FUNCTION_BLOCK FB_RecipeBase IMPLEMENTS I_RecipeBuilder 

VAR
    _Config                 : ST_RecipeBuilder_Config;
	_ConfigProvider 		: I_GantryConfigProvider;

	
	
	_Limits : ST_Recipe_Limits;

    // --- NOWE ZMIENNE DO PRZECHOWYWANIA SEGMENTÓW ---
    _SegmentsCutX           : ARRAY [1..100] OF ST_CutSegment;
    _SegmentsCutY           : ARRAY [1..100] OF ST_CutSegment;
    _SegmentsGroove         : ARRAY [1..100] OF ST_CutSegment;
	_HolesDrill 			: ARRAY [1..100] OF ST_PointXY;
	_ShapeStart         	: ARRAY [1..100] OF ST_PointXY;
	_ShapesCount        	: INT := 1;
    _CurrentShapeIndex  	: INT := 1;
	_HolesToDrill   		: INT;
    _SegmentsToCutX         : INT;
    _SegmentsToCutY         : INT;
    _SegmentsToGroove       : INT;
	_FootprintX 			: REAL;
	_FootprintY 			: REAL;
	_MaxCopiesX				: DINT;
	_MaxCopiesY				: DINT;
	_ActualCopiesX			: DINT;
	_ActualCopiesY			: DINT;
	_NominalX 				: REAL;
    _NominalY 				: REAL;
	_Busy					: BOOL;
	_Done					: BOOL;
	_Error					: BOOL;
	
	// --- GENERYCZNY GENERATOR G-CODE (NCI) ---
    fbCreateFile    : ItpPpgCreateMain;
    fbAppendLine    : ItpPpgAppendGenericBlock;
    fbCloseFile     : ItpPpgCloseMain;
    
    _aGCodeBuffer   : ARRAY[1..600] OF STRING(255); 
    _nLinesToWrite  : INT;                          // Ile linii z bufora zapisać
    _nFileWriteStep : INT := 0;                     // Krok maszyny stanów zapisu
    _sGCodeFilePath : STRING(255);                  // Ścieżka pliku
	
	_GeometryWriter : I_GeometryWriter;
	
END_VAR

PROPERTY ActualCopiesX : DINT
GET
ActualCopiesX := _Config.RequestedCopiesX;
END_GET
END_PROPERTY

PROPERTY ActualCopiesY : DINT
GET
ActualCopiesY := _Config.RequestedCopiesY;
END_GET
END_PROPERTY

METHOD Build : BOOL
Build := FALSE;
END_METHOD

PROPERTY Busy : BOOL
GET
Busy := _Busy;
END_GET
SET
_Busy := Busy;
END_SET
END_PROPERTY

METHOD PROTECTED CalculateFootprint
VAR_INPUT
END_VAR
// Domyślny wymiar detalu (bez dodatków)
_NominalX := _Config.PanelFrontWidth;
_NominalY := _Config.PanelFrontLength;
END_METHOD

PROPERTY Config : ST_RecipeBuilder_Config
GET
Config := _Config;
END_GET
SET
VAR
    sTempGCodePath : STRING(255);
END_VAR
// 1. NAJPIERW robimy kopię tego co mamy w pamięci sterownika
sTempGCodePath := THIS^._Config.GCodePath; 

// 2. TERAZ przyjmujemy nową strukturę z HMI
_Config := Config;

// 3. PRZYWRACAMY ścieżkę do pliku
_Config.GCodePath := sTempGCodePath;

_Config.PanelFrontLength     := LIMIT(_Limits.PanelFrontLength.MinVal, Config.PanelFrontLength, _Limits.PanelFrontLength.MaxVal);
_Config.PanelFrontWidth      := LIMIT(_Limits.PanelFrontWidth.MinVal,  Config.PanelFrontWidth,  _Limits.PanelFrontWidth.MaxVal);
_Config.PanelHeight          := LIMIT(_Limits.PanelHeight.MinVal,      Config.PanelHeight,      _Limits.PanelHeight.MaxVal);
_Config.RailHeightCorrection := LIMIT(_Limits.RailHeightCorrection.MinVal, Config.RailHeightCorrection, _Limits.RailHeightCorrection.MaxVal);
_Config.GrooveDepthZ		 :=	LIMIT(_Limits.GrooveDepthZ.MinVal,	Config.GrooveDepthZ, _Limits.GrooveDepthZ.MaxVal);
_Config.Diameter 			 := LIMIT(_Limits.Diameter.MinVal, Config.Diameter, _Limits.Diameter.MaxVal);

_Config.CuttingOverpass      := LIMIT(_Limits.CuttingOverpass.MinVal, Config.CuttingOverpass, _Limits.CuttingOverpass.MaxVal);
_Config.GroovingOverpass     := LIMIT(_Limits.GroovingOverpass.MinVal, Config.GroovingOverpass, _Limits.GroovingOverpass.MaxVal);
_Config.Radius               := LIMIT(_Limits.Radius.MinVal, Config.Radius, _Limits.Radius.MaxVal);

THIS^.UpdateNestingLimits();


IF _Config.FillAll THEN
    _Config.RequestedCopiesX := _MaxCopiesX;
    _Config.RequestedCopiesY := _MaxCopiesY;
ELSE
    _Config.RequestedCopiesX := LIMIT(1, _Config.RequestedCopiesX, _MaxCopiesX);
    _Config.RequestedCopiesY := LIMIT(1, _Config.RequestedCopiesY, _MaxCopiesY);
END_IF
END_SET
END_PROPERTY

PROPERTY ConfigProvider : I_GantryConfigProvider
GET
ConfigProvider := _ConfigProvider;
END_GET
SET
_ConfigProvider := ConfigProvider;
END_SET
END_PROPERTY

PROPERTY CurrentShapeIndex : INT
GET
CurrentShapeIndex := _CurrentShapeIndex;
END_GET
SET
_CurrentShapeIndex := CurrentShapeIndex;
END_SET
END_PROPERTY

PROPERTY Done : BOOL
GET
Done := _Done;
END_GET
SET
_Done := Done;
END_SET
END_PROPERTY

PROPERTY Error : BOOL
GET
Error := _Error;
END_GET
SET
_Error := Error;
END_SET
END_PROPERTY

PROPERTY ExecutionRoute : E_ExecutionRoute
GET
END_GET
END_PROPERTY

PROPERTY FootprintX : REAL
GET
FootprintX := _FootprintX;
END_GET
SET
_FootprintX := FootprintX;
END_SET
END_PROPERTY

PROPERTY FootprintY : REAL
GET
FootprintY := _FootprintY;
END_GET
SET
_FootprintY := FootprintY;
END_SET
END_PROPERTY

PROPERTY GeometryWriter : I_GeometryWriter
GET
GeometryWriter := _GeometryWriter;
END_GET
SET
_GeometryWriter := GeometryWriter;
END_SET
END_PROPERTY

PROPERTY HolesDrill : REFERENCE TO ARRAY [1..100] OF ST_PointXY
GET
HolesDrill REF= _HolesDrill;
END_GET
END_PROPERTY

PROPERTY HolesToDrill : INT
GET
HolesToDrill := _HolesToDrill;
END_GET
END_PROPERTY

PROPERTY Limits : ST_Recipe_Limits
GET
Limits := _Limits;
END_GET
END_PROPERTY

PROPERTY MaxCopiesX : DINT
GET
MaxCopiesX := _MaxCopiesX;
END_GET
END_PROPERTY

PROPERTY MaxCopiesY : DINT
GET
MaxCopiesY := _MaxCopiesY ;
END_GET
END_PROPERTY

PROPERTY SegmentsCutX : REFERENCE TO ARRAY [1..100] OF ST_CutSegment
GET
SegmentsCutX REF= _SegmentsCutX;
END_GET
END_PROPERTY

PROPERTY SegmentsCutY : REFERENCE TO ARRAY [1..100] OF ST_CutSegment
GET
SegmentsCutY REF= _SegmentsCutY;
END_GET
END_PROPERTY

PROPERTY SegmentsGroove : REFERENCE TO ARRAY [1..100] OF ST_CutSegment
GET
SegmentsGroove REF= _SegmentsGroove;
END_GET
END_PROPERTY


PROPERTY SegmentsToCutX : INT
GET
SegmentsToCutX := _SegmentsToCutX;
END_GET
END_PROPERTY


PROPERTY SegmentsToCutY : INT
GET
SegmentsToCutY := _SegmentsToCutY;
END_GET
END_PROPERTY


PROPERTY SegmentsToGroove : INT
GET
SegmentsToGroove := _SegmentsToGroove;
END_GET
END_PROPERTY

PROPERTY ShapesCount : INT
GET
ShapesCount := _ShapesCount;
END_GET
END_PROPERTY

PROPERTY ShapeStart : REFERENCE TO ARRAY [1..100] OF ST_PointXY
GET
ShapeStart REF= _ShapeStart;
END_GET
END_PROPERTY

METHOD PUBLIC UpdateNestingLimits
VAR
    MaxOverpass     : REAL;
    MachineConfig   : ST_GantryXYZ_Config; // Zmienna do odczytu offsetu
    EffectiveBoardX : REAL;
    EffectiveBoardY : REAL;
END_VAR
VAR_INST
    bLogFired       : BOOL; // <-- Zapamięta, czy log już poszedł
END_VAR
// 1. Czysty gabaryt z logiki receptury
THIS^.CalculateFootprint();
MaxOverpass := MAX(_Config.CuttingOverpass, _Config.GroovingOverpass);
_FootprintX := _NominalX + (2.0 * MaxOverpass);
_FootprintY := _NominalY + (2.0 * MaxOverpass);

// 2. Pobranie Global Offsetu ORAZ wymiarów płyty z maszyny
IF _ConfigProvider <> 0 THEN
    MachineConfig := _ConfigProvider.Config;
ELSE
    // Awaryjny "fallback" jeśli Provider nie jest wstrzyknięty (np. w starych testach)
    MachineConfig.GlobalOffsetX := 0.0;
    MachineConfig.GlobalOffsetY := 0.0;
    MachineConfig.RawBoardX := 1220.0; // Domyślna płyta 
    MachineConfig.RawBoardY := 2440.0; // Domyślna płyta
	MachineConfig.RawBoardZ := 9.0;
END_IF

// 3. Efektywna wielkość płyty = Fizyczna płyta (z maszyny) minus offset początkowy
EffectiveBoardX := MachineConfig.RawBoardX - MachineConfig.GlobalOffsetX;
EffectiveBoardY := MachineConfig.RawBoardY - MachineConfig.GlobalOffsetY;

// 4. Przeliczanie kopii nestingu (zabezpieczenie na ujemne wymiary)
IF _FootprintX > 0.0 AND EffectiveBoardX > 0.0 THEN
    _MaxCopiesX := REAL_TO_DINT(TRUNC(EffectiveBoardX / _FootprintX));
ELSE
    _MaxCopiesX := 0;
END_IF

IF _FootprintY > 0.0 AND EffectiveBoardY > 0.0 THEN
    _MaxCopiesY := REAL_TO_DINT(TRUNC(EffectiveBoardY / _FootprintY));
ELSE
    _MaxCopiesY := 0;
END_IF

// =========================================================
// 5. WERYFIKACJA GABARYTÓW (Zabezpieczenie przed za dużym detalem)
// =========================================================
_Config.IsValid := (_MaxCopiesX > 0) AND (_MaxCopiesY > 0) AND (_NominalX > 0) AND (_NominalY > 0);

IF NOT _Config.IsValid THEN
    IF NOT bLogFired THEN
        ADSLOGSTR(ADSLOG_MSGTYPE_ERROR, 'UpdateNestingLimits: Konfiguracja odrzucona (IsValid = FALSE)! Sprawdzam dlaczego...', '');
        
        IF _MaxCopiesX <= 0 THEN 
            ADSLOGSTR(ADSLOG_MSGTYPE_ERROR, 'Powod: _MaxCopiesX <= 0 (Detal wychodzi poza szerokosc stolu)', ''); 
        END_IF
        IF _MaxCopiesY <= 0 THEN 
            ADSLOGSTR(ADSLOG_MSGTYPE_ERROR, 'Powod: _MaxCopiesY <= 0 (Detal wychodzi poza dlugosc stolu)', ''); 
        END_IF
        IF _NominalX <= 0 THEN 
            ADSLOGSTR(ADSLOG_MSGTYPE_ERROR, 'Powod: _NominalX <= 0 (Szerokosc Nominalna to zero!)', ''); 
        END_IF
        IF _NominalY <= 0 THEN 
            ADSLOGSTR(ADSLOG_MSGTYPE_ERROR, 'Powod: _NominalY <= 0 (Dlugosc Nominalna to zero!)', ''); 
        END_IF
        
        bLogFired := TRUE; // Zablokuj kolejne wysyłanie
    END_IF
ELSE
    // Jeśli znowu jest poprawnie (np. poprawiono na HMI), odblokuj logi na przyszłość
    bLogFired := FALSE;
END_IF

// =========================================================
// 6. AUTO-KOREKTA KOPII I LIMITÓW DLA HMI
// =========================================================

// ZABEZPIECZENIE Z: Głębokość frezowania nie może przekroczyć grubości płyty!
_Limits.GrooveDepthZ.MaxVal := MachineConfig.RawBoardZ + 4.0;
// Bezlitosne obcięcie (clamping) wpisanej wartości do nowego limitu
_Config.GrooveDepthZ := LIMIT(_Limits.GrooveDepthZ.MinVal, _Config.GrooveDepthZ, _Limits.GrooveDepthZ.MaxVal);

IF _Config.IsValid THEN
    _Limits.RequestedCopiesX.MinVal := 1.0;
    _Limits.RequestedCopiesX.MaxVal := DINT_TO_REAL(_MaxCopiesX);
    _Limits.RequestedCopiesY.MinVal := 1.0;
    _Limits.RequestedCopiesY.MaxVal := DINT_TO_REAL(_MaxCopiesY);

    IF _Config.FillAll THEN
        _Config.RequestedCopiesX := _MaxCopiesX;
        _Config.RequestedCopiesY := _MaxCopiesY;
    ELSE
        _Config.RequestedCopiesX := LIMIT(1, _Config.RequestedCopiesX, _MaxCopiesX);
        _Config.RequestedCopiesY := LIMIT(1, _Config.RequestedCopiesY, _MaxCopiesY);
    END_IF
ELSE
    // Blokada całkowita jeśli detal się nie mieści
    _Limits.RequestedCopiesX.MinVal := 0.0;
    _Limits.RequestedCopiesX.MaxVal := 0.0;
    _Limits.RequestedCopiesY.MinVal := 0.0;
    _Limits.RequestedCopiesY.MaxVal := 0.0;
    
    _Config.RequestedCopiesX := 0;
    _Config.RequestedCopiesY := 0;
END_IF
END_METHOD

METHOD PROTECTED WriteGCodeFile : BOOL
VAR_INPUT
    sFilePath : STRING(255);
END_VAR
VAR_INST
	_iCurrentLine : INT := 1;
END_VAR
WriteGCodeFile := FALSE;

CASE _nFileWriteStep OF
    0: // INIT
        _iCurrentLine := 1; 
        _sGCodeFilePath := sFilePath;
        
        // LOG: Start operacji - wstawiamy zmienną string w miejsce %s
        ADSLOGSTR(ADSLOG_MSGTYPE_HINT, 'WriteGCode: Rozpoczynam zapis do pliku %s', _sGCodeFilePath);
        
        _nFileWriteStep := 10;

    10: // --- OTWIERANIE/TWORZENIE PLIKU ---
        fbCreateFile(
            bExecute := TRUE, 
            sPathName := _sGCodeFilePath, 
            tTimeOut := T#2S
        );
        
        IF fbCreateFile.bErr THEN 
            // LOG: Błąd tworzenia
            ADSLOGSTR(ADSLOG_MSGTYPE_ERROR, 'WriteGCode: BLAD tworzenia pliku %s!', _sGCodeFilePath);
            _nFileWriteStep := 999;
            
        ELSIF NOT fbCreateFile.bBusy THEN
            fbCreateFile(bExecute := FALSE, sPathName := _sGCodeFilePath);
            
            // LOG: Sukces tworzenia
            ADSLOGSTR(ADSLOG_MSGTYPE_HINT, 'WriteGCode: Plik utworzony pomyslnie, przechodze do zapisu.', '');
            _nFileWriteStep := 20;
        END_IF

    20: // --- ZAPISYWANIE LINII G-CODE W PĘTLI ---
        fbAppendLine(
            bExecute := TRUE, 
            sPathName := _sGCodeFilePath, 
            sBlock := _aGCodeBuffer[_iCurrentLine], 
            tTimeOut := T#2S
        );
        
        IF fbAppendLine.bErr THEN 
            // LOG: Błąd zapisu konkretnej linii
            ADSLOGSTR(ADSLOG_MSGTYPE_ERROR, 'WriteGCode: BLAD dopisywania linii G-Code!', '');
            _nFileWriteStep := 999;
            
        ELSIF NOT fbAppendLine.bBusy THEN
            fbAppendLine(bExecute := FALSE, sPathName := _sGCodeFilePath);
            
            _iCurrentLine := _iCurrentLine + 1;
            IF _iCurrentLine > _nLinesToWrite THEN
                // LOG: Koniec pętli zapisu
                ADSLOGSTR(ADSLOG_MSGTYPE_HINT, 'WriteGCode: Zapisano wszystkie linie G-Code.', '');
                _nFileWriteStep := 30; // Zapisano wszystkie linie
            END_IF
        END_IF

    30: // --- ZAMYKANIE PLIKU ---
        fbCloseFile(
            bExecute := TRUE, 
            sPathName := _sGCodeFilePath, 
            tTimeOut := T#2S
        );
        
        IF fbCloseFile.bErr THEN 
            // LOG: Błąd zamykania
            ADSLOGSTR(ADSLOG_MSGTYPE_ERROR, 'WriteGCode: BLAD zamykania pliku!', '');
            _nFileWriteStep := 999;
            
        ELSIF NOT fbCloseFile.bBusy THEN
            fbCloseFile(bExecute := FALSE, sPathName := _sGCodeFilePath);
            
            // Zapisujemy ścieżkę do struktury Config, żeby Executor NCI wiedział co odpalić
            _Config.GCodePath := _sGCodeFilePath; 
            
            // LOG: Pełny sukces
            ADSLOGSTR(ADSLOG_MSGTYPE_HINT, 'WriteGCode: Plik zamkniety pomyslnie.', '');
            _nFileWriteStep := 1000;
        END_IF

    999: // --- BŁĄD ---
        WriteGCodeFile := FALSE;
        // W tym kroku nie dajemy loga, zeby nie zaspamować konsoli błędem co każdy cykl!
        // Logi błędu wysłaliśmy tuż przed przejściem do kroku 999.

    1000: // --- GOTOWE ---
        _nFileWriteStep := 0; // Reset na przyszłość
        WriteGCodeFile := TRUE;
        
END_CASE
END_METHOD

END_FUNCTION_BLOCK

(* stored: Version 1.1.0.1, ProductVersion 3.1.4024.15
   POU FB_RecipeBase: Id {da96ec31-8163-452f-a094-4558fa21ef5c}, SpecialFunc None
   Property ActualCopiesX: Id {f6bb53f7-fe6a-4e43-854b-3965a8a4a1af}
   Get Get: Id {acf86470-a159-4078-98de-d4ec1d0fe9ea}
   Property ActualCopiesY: Id {28c47b7e-b948-4a5e-8a09-4953e885c928}
   Get Get: Id {0f5cef6e-b24f-4a80-ae1b-1e315e1a7393}
   Method Build: Id {47409b61-265d-42e6-ab22-9bedebae5b88}
   Property Busy: Id {a9db9b6c-8eb1-4c93-8b62-2f01d1c13c3a}
   Get Get: Id {483f8e7b-8254-4848-b7d1-613795426f51}
   Set Set: Id {1243a542-e270-4a34-813e-02853c7e0109}
   Method CalculateFootprint: Id {b5903cf0-35f3-4a36-9bbd-0a6781b9e2f5}
   Property Config: Id {cc8b22ea-aed1-438f-8cdd-5e3e5f7b2e90}
   Get Get: Id {51a4be92-27e0-4d30-897e-f466d704a9e2}
   Set Set: Id {ea17f2c2-4fb3-4cd4-85eb-6bcadc1e2873}
   Property ConfigProvider: Id {8b0de6b1-3957-44a3-88b0-341b09b0b39a}
   Get Get: Id {2167364a-f1be-4cf1-9920-cef8a1292a7b}
   Set Set: Id {2269ab13-305f-4ee2-8020-24ff434eedbe}
   Property CurrentShapeIndex: Id {26917ea1-1cef-41af-a616-e7c3bffaf80f}
   Get Get: Id {2e3bb86d-b7ac-4e77-8962-142bcaba5f0e}
   Set Set: Id {d4715697-fd64-40db-8769-f30824d5d94b}
   Property Done: Id {95f7dd68-43a4-412e-aee7-bfaa1fc7a303}
   Get Get: Id {f917eb4b-8c90-4223-a28c-4f44be300935}
   Set Set: Id {e5ea673e-d2a8-4e8f-9caf-1b2230715dca}
   Property Error: Id {5a010892-cf00-4d6b-a054-1dc9b83bd5cd}
   Get Get: Id {c1aca7d3-ffa8-424c-8a8a-0100db86b490}
   Set Set: Id {41b517d7-5e51-4abd-a86d-80b23eeef3ea}
   Property ExecutionRoute: Id {d2212b52-9f21-4298-b628-266a7518ecb2}
   Get Get: Id {8041d254-a158-4e66-a29b-c43d3e45cbc2}
   Property FootprintX: Id {31cc2579-4943-4072-adcb-7298a1ade9ce}
   Get Get: Id {e9997c45-4a9f-41c6-91e6-e1fa92e42836}
   Set Set: Id {4b7b29b6-122d-49af-a98f-be17039311b8}
   Property FootprintY: Id {ff2a3b37-b1bb-44a6-b5de-6e4f50f25550}
   Get Get: Id {7db99de3-36d4-4fef-ac1d-4a0b509bbfca}
   Set Set: Id {28566d1d-285b-4a14-82b8-bb0c44370488}
   Property GeometryWriter: Id {0595b86d-12dc-4c63-b408-5e7e23b5a0e1}
   Get Get: Id {e798f707-68ae-4415-b903-6eaef2d95e9e}
   Set Set: Id {c0543439-b8f5-43b2-aaf0-f68e18613a3b}
   Property HolesDrill: Id {33a6c722-63d3-4021-9875-0f4e89b1bc5f}
   Get Get: Id {353ebf4d-ee7a-4628-96f6-0d8b60355f97}
   Property HolesToDrill: Id {0da1219c-5551-48b2-8898-9bdf935c4a67}
   Get Get: Id {98d6479b-e543-4802-b7d4-dfa0834b198e}
   Property Limits: Id {d6f83e87-8dd7-4840-949b-411b575caaa2}
   Get Get: Id {ec01404a-7a39-4271-9193-9e9005040333}
   Property MaxCopiesX: Id {141e0a02-d648-49f9-a7cf-0bb7a2866c40}
   Get Get: Id {01ae6afa-0069-4c7f-a7d7-529c551d837a}
   Property MaxCopiesY: Id {020d58bf-374a-498a-a7f1-941fa55b76a6}
   Get Get: Id {34530db3-9b5f-4311-bde6-21781e13e93c}
   Property SegmentsCutX: Id {3184be54-f03a-4975-8cf1-db07c128d253}
   Get Get: Id {0f425160-36a8-4f28-99b9-e92bc5ef61d9}
   Property SegmentsCutY: Id {7e96d748-34eb-4d02-bea9-39c6162fca26}
   Get Get: Id {18ebbd77-7872-47d5-b7ea-e1c19856104e}
   Property SegmentsGroove: Id {ef32f872-b41e-411a-89df-3b90001a16fb}
   Get Get: Id {9f573555-28d1-42d5-8de5-c6e1c98b00d0}
   Property SegmentsToCutX: Id {7c141887-7a79-44a8-a421-fb9ee098c25b}
   Get Get: Id {549e99d8-5984-4542-b902-6ce577ebde0d}
   Property SegmentsToCutY: Id {2a1a5acb-e3ff-4cf0-ad15-d0b6b45a1d0e}
   Get Get: Id {4f78cbac-d000-4132-997b-ee432b29e987}
   Property SegmentsToGroove: Id {c7b518f5-2d21-49fc-94c1-1f117859a4b1}
   Get Get: Id {8e366a6f-311d-4e3a-904c-a58ce6da4751}
   Property ShapesCount: Id {ddd120b9-00cd-4b1c-b2b1-0fde6185de6f}
   Get Get: Id {f3cff4d1-f4e1-44c8-8b4a-4d472803af48}
   Property ShapeStart: Id {52d57a51-14a0-4aab-abe9-db16b054b96d}
   Get Get: Id {130de704-36d0-4d0c-80da-43de01c2c5c4}
   Method UpdateNestingLimits: Id {b78c73fe-7983-4c8d-9c71-a0293b8dccf5}
   Method WriteGCodeFile: Id {b115e39c-0872-441f-a4ac-20c73a4f870f} *)
